Universal Robots PolyScope program: d_to_a.urp

Program d_to_a (installation=string_planes directory=/programs createdIn=5.17.3 lastSavedIn=5.17.3 robotSerialNumber=20245501435)
Calibrated DH parameters: a=[0.000154, -0.137004, -0.385524, -0.00002, 0.000092, 0]; d=[0.162441, 211.794786, -230.585024, 18.923638, 0.099786, 0.09951]; alpha=[1.569493, -0.001902, 0.003874, 1.570111, -1.570167, 0]; deltaTheta=[0, -1.242934, 1.056292, 0.186646, 0.000002, 0.000001]
InitVariablesNode
Robot Program (runOnlyOnce=false)
  MoveJ speed 60 deg/s, acceleration 80 deg/s^2 (useActiveTCP=true) feature=Base
    Waypoint Waypoint_1 (Relative): relativeFromPosition TCP in base x=337.271 y=452.585 z=146.267 mm, rx=-1.6083 ry=-2.1977 rz=1.0429 rad; joints [-146.226, -47.168, 100.749, -99.801, -91.439, -163.024] deg; TCP offset x=28.21 y=-96.107 z=-99.69 mm, rx=0 ry=0 rz=0 rad; TCP in base x=327.38 y=541.714 z=231.884 mm, rx=1.6818 ry=2.3248 rz=-1.1114 rad; joints [-139.64, -50.321, 85.996, -84.697, -102.358, -153.08] deg
